(* IEC 61131-3 sources: learning-path/05_oop_in_st/exercises/4_inheritance_complex_valve/src, 3 files *)

(* ---- TankStates.st ---- *)
NAMESPACE FluidHandlingClass
    TYPE
        TankState : (Filling, Emptying, Flushing, Close) := Close;
    END_TYPE
END_NAMESPACE

(* ---- configuration.st ---- *)
USING FluidHandlingClass;
CONFIGURATION MyConfiguration
    TASK Main(Interval := T#1000ms, Priority := 1);
    PROGRAM P1 WITH Main: CalculatorCurrentVolume;
    VAR_GLOBAL

        //FIRST IMPLEMENTATION SIMPLE
        vIn : basicValve;
        vOut: basicValveValve;
        tank : TankWithVolume := (inletValve := vIn, outletValve := vOut, volume := 100);

        //SIMPLE VALVES
        vInCtrl AT %Q1.0 : BOOL;
        vOutCtrl AT %Q1.1 : BOOL;

        vInOpen : BOOL;
        vOutOpen : BOOL;
        vInClosed : BOOL;
        vOutClosed : BOOL;

        statusIn : ValveState;
        statusOut : ValveState;

        //CONTROL TANK
        Close AT %I0.0 : BOOL;
        Fill AT %I0.1  : BOOL;
        Empty AT %I0.2 : BOOL;
        Flush AT %I0.3  : BOOL;
        phase : TankState;
    END_VAR
END_CONFIGURATION

(* ---- program.st ---- *)
USING FluidHandlingClass;
USING System.Timer;

// Imagine that the filling rate is 5 L/s when the inlet valve is Open

PROGRAM CalculatorCurrentVolume
    VAR_EXTERNAL
        vIn  : Valve2;
        vOut : Valve2;
        tank : TankWithVolume;

        vInCtrl  : BOOL;
        vOutCtrl : BOOL;

        vInOpen : BOOL;
        vOutOpen : BOOL;
        vInClosed : BOOL;
        vOutClosed : BOOL;
        statusIn : ValveState;
        statusOut : ValveState;

        Close : BOOL;
        Fill  : BOOL;
        Empty : BOOL;
        Flush : BOOL;
        phase : TankState;
    END_VAR
    VAR
        _ton : OnDelay := (duration := T#1s);
        _duration_max  : LTIME;
        current_volume : REAL := 0;
        capacity_percentage : REAL;
        _filling_rate : REAL;
        _emptying_rate: REAL;

    END_VAR
    _ton();
    _duration_max :=  TO_LTIME(TO_LINT(tank.volume / 5));  //Conversion to Time values
    _filling_rate := 1;  //LATER EXPRESION WITH THE OPENING/CLOSING RATES
    _emptying_rate := 1; //SAME AS FILLING RATE
    capacity_percentage := tank.Capacity(currentVolume := current_volume);
    statusIn := vIn.GetState();
    statusOut := vOut.GetState();
    tank.ReadCyclic(Fill := Fill, Empty := Empty, Flush := Flush,  Close := Close);

    CASE phase OF
        //-----------------------------------
        // here's the tank phase close
        //-----------------------------------

            TankState#Close:
            tank.Close();
            IF (Fill) THEN
                _ton.signal := TRUE;
                phase := TankState#Filling;
            END_IF;
            IF (Empty) THEN
                _ton.signal := TRUE;
                phase:= TankState#Emptying;
            END_IF;
            IF (Flush) THEN
                _ton.signal := TRUE;
                phase := TankState#Flushing;
            END_IF;
            // next phase after timeout

        //-----------------------------------
        // here's the tank phase Filling
        //-----------------------------------
        TankState#Filling:

            // next phase after timeout
            IF (Fill) THEN
                tank.Fill();
                IF (capacity_percentage > 100) THEN
                    _ton.signal := FALSE;
                    phase := TankState#Close;
                END_IF;
                IF _ton.output THEN
                    _ton.signal := FALSE;
                    current_volume := current_volume + 5 *_filling_rate; //Increment the volume in 5 Liters per second
                    IF current_volume > tank.volume THEN
                        current_volume := tank.volume; //Ensure volume does not exceed the maximum volume
                    END_IF;
                    capacity_percentage := tank.Capacity(currentVolume := current_volume);; // Actualize the capacity percentage
                    _ton.signal := TRUE; // Reinitialice the timer
                END_IF;

            ELSE
                _ton.signal := FALSE;
                phase := TankState#Close;
            END_IF;
        //-----------------------------------
        // here's the tank phase Emptying
        //-----------------------------------
        TankState#Emptying:
            IF (Empty) THEN
                tank.Emptying();
                IF (capacity_percentage <= 0) THEN
                    _ton.signal := FALSE;
                    phase := TankState#Close;
                END_IF;
                IF _ton.output THEN
                    _ton.signal := FALSE;
                    current_volume := current_volume - 5 *_emptying_rate; //Reduce the volume in 5 Liters per second
                    IF current_volume < 0 THEN
                        current_volume := 0; // //Ensure volume does not exceed the minimum volume
                    END_IF;
                    END_IF;
                    capacity_percentage := tank.Capacity(currentVolume := current_volume);; //Actualize the capacity percentage
                    _ton.signal := TRUE; // Reinitialice the timer
                END_IF;

            ELSE
                _ton.signal := FALSE;
                phase := TankState#Close;
            END_IF;
        //-----------------------------------
        // here's the tank phase Flushing (HERE THAT THE FILLING AND EMPTYING RATE IS THE SAME DOESN'T DO ANYTHING)
        //-----------------------------------
        TankState#Flushing:
            IF Flush THEN
                tank.Flush();
                _ton.signal := TRUE;

            ELSE
                _ton.signal := FALSE;
                phase := TankState#Close;
            END_IF;
    END_CASE;

    vIn.WriteCyclic(ctrlOpen => vInCtrl, isOpen => vInOpen, isClosed => vInClosed, state => statusIn);
    vOut.WriteCyclic(ctrlOpen => vOutCtrl, isOpen => vOutOpen, isClosed => vOutClosed, state => statusOut);
    tank.WriteCyclic(Capacity => capacity_percentage);
END_PROGRAM
